(* IEC 61131-3 sources: moqui-plc/iec61131/moqui/framework/src/main/org/moqui/device, 53 files *)

(* ---- ActuatorActuationType.dut ---- *)
(*#-#-#-#-#-#-#-#-#-#---Declaration---#-#-#-#-#-#-#-#-#-#-#-#-#*)

{attribute 'qualified_only'}
{attribute 'strict'}
TYPE ActuatorActuationType : (
    SingleActuation := 0, (* Single Actuation: Uses enable output only *)
    DoubleActuation, (* Double Actuation: enable/disable are pulses *)
    DoubleActuationNoRetain (* Double Actuation: enable/disable are levels *)
); END_TYPE

(* ---- ActuatorActuationType.st ---- *)
TYPE ActuatorActuationType : (
    SingleActuation := 0, (* Single Actuation: Uses enable output only *)
    DoubleActuation, (* Double Actuation: enable/disable are pulses *)
    DoubleActuationNoRetain (* Double Actuation: enable/disable are levels *)
); END_TYPE

(* ---- ActuatorFeedbackType.dut ---- *)
(*#-#-#-#-#-#-#-#-#-#---Declaration---#-#-#-#-#-#-#-#-#-#-#-#-#*)

{attribute 'qualified_only'}
{attribute 'strict'}
TYPE ActuatorFeedbackType : (
	WithoutFeedback := 0, (* No feedback *)
    SingleDisableFeedback, (* Single Deactivation Feedback: Only disabledSensor *)
    SingleEnableFeedback, (* Single Activation Feedback: Only enabledSensor *)
	DoubleFeedback (* Double Feedback: Both sensors *)
); END_TYPE

(* ---- ActuatorFeedbackType.st ---- *)
TYPE ActuatorFeedbackType : (
	WithoutFeedback := 0, (* No feedback *)
    SingleDisableFeedback, (* Single Deactivation Feedback: Only disabledSensor *)
    SingleEnableFeedback, (* Single Activation Feedback: Only enabledSensor *)
	DoubleFeedback (* Double Feedback: Both sensors *)
); END_TYPE

(* ---- ActuatorGroupAutochange.dut ---- *)
(*#-#-#-#-#-#-#-#-#-#---Declaration---#-#-#-#-#-#-#-#-#-#-#-#-#*)

{attribute 'qualified_only'}
{attribute 'strict'}
(*
 * Selects the mode used to trigger a priority-order rotation (autochange).
 * Corresponds to ABB ACH580 parameter 76.70 Autochange.
 *)
TYPE ActuatorGroupAutochange : (
    None := 0, (* Autochange disabled; priority order is fixed *)
    EvenWear, (* Rotate when run-hour imbalance > maxWearImbalance (76.72) *)
    FixedInterval, (* Rotate every autochangeInterval when demand ≤ autochangeLevel (76.71) *)
    ExternalTrigger, (* Rotate on rising edge of autochangeTrigger when demand ≤ autochangeLevel *)
    AllStopped (* Rotate whenever the group stops (all actuators off) *)
); END_TYPE

(* ---- ActuatorGroupAutochange.st ---- *)
(*
 * Selects the mode used to trigger a priority-order rotation (autochange).
 * Corresponds to ABB ACH580 parameter 76.70 Autochange.
 *)
TYPE ActuatorGroupAutochange : (
    None := 0, (* Autochange disabled; priority order is fixed *)
    EvenWear, (* Rotate when run-hour imbalance > maxWearImbalance (76.72) *)
    FixedInterval, (* Rotate every autochangeInterval when demand <= autochangeLevel (76.71) *)
    ExternalTrigger, (* Rotate on rising edge of autochangeTrigger when demand <= autochangeLevel *)
    AllStopped (* Rotate whenever the group stops (all actuators off) *)
); END_TYPE

(* ---- ActuatorGroupStatus.dut ---- *)
(*#-#-#-#-#-#-#-#-#-#---Declaration---#-#-#-#-#-#-#-#-#-#-#-#-#*)

{attribute 'qualified_only'}
{attribute 'strict'}
TYPE ActuatorGroupStatus : (
    Disabled := 0, (* No actuators running; group not active *)
    Running, (* Active: demand-driven start/stop in progress *)
    Stopping, (* Transitional: shutting down all running actuators *)
    Autochange (* Transitional: rotating the priority order (stop old / start new) *)
); END_TYPE

(* ---- ActuatorGroupStatus.st ---- *)
TYPE ActuatorGroupStatus : (
    Disabled := 0, (* No actuators running; group not active *)
    Running, (* Active: demand-driven start/stop in progress *)
    Stopping, (* Transitional: shutting down all running actuators *)
    Autochange (* Transitional: rotating the priority order (stop old / start new) *)
); END_TYPE

(* ---- ActuatorModel.dut ---- *)
(*#-#-#-#-#-#-#-#-#-#---Declaration---#-#-#-#-#-#-#-#-#-#-#-#-#*)

{attribute 'qualified_only'}
TYPE ActuatorModel : (
	ABBACH580, (* ABB ACH580 *)
	CTM700, (* Control Techniques CM700 *)
	DanfossFC102, (* Danfoss FC102 *)
	ABBPSTX (* ABB PSTX SoftStarter *)
	(* etc. *)
); END_TYPE

(* ---- ActuatorStatus.dut ---- *)
(*#-#-#-#-#-#-#-#-#-#---Declaration---#-#-#-#-#-#-#-#-#-#-#-#-#*)

{attribute 'qualified_only'}
{attribute 'strict'}
TYPE ActuatorStatus : (
	Disabled := 0, (* Stable *)
	EnablePhase, (* Unstable *)
	Enabled, (* Stable *)
	DisablePhase (* Unstable *)
); END_TYPE

(* ---- ActuatorStatus.st ---- *)
TYPE ActuatorStatus : (
	Disabled := 0, (* Stable *)
	EnablePhase, (* Unstable *)
	Enabled, (* Stable *)
	DisablePhase (* Unstable *)
); END_TYPE

(* ---- ActuatorType.dut ---- *)
(*#-#-#-#-#-#-#-#-#-#---Declaration---#-#-#-#-#-#-#-#-#-#-#-#-#*)

{attribute 'qualified_only'}
{attribute 'strict'}
TYPE ActuatorType : (
  OnOff := 0, (* Fallback value *)
  Contactor,
  SoftStarter,
  Vfd, (* Frequency converter / Inverter drive *)
  PneumaticCylinder,
  PneumaticValve,
  HydraulicCylinder,
  HydraulicValve,
  Damper,
  SolenoidValve
  (* etc. *)
); END_TYPE

(* ---- ActuatorType.st ---- *)
TYPE ActuatorType : (
  OnOff := 0, (* Fallback value *)
  Contactor,
  SoftStarter,
  Vfd, (* Frequency converter / Inverter drive *)
  PneumaticCylinder,
  PneumaticValve,
  HydraulicCylinder,
  HydraulicValve,
  Damper,
  SolenoidValve
  (* etc. *)
); END_TYPE

(* ---- DeviceConfigCmdType.dut ---- *)
(*#-#-#-#-#-#-#-#-#-#---Declaration---#-#-#-#-#-#-#-#-#-#-#-#-#*)

{attribute 'qualified_only'}
{attribute 'strict'}
(* After each creation, saving or deletion of device config it will be necessary to reload the config list with the Init command. *)
TYPE DeviceConfigCmdType : (
    Init := 0, (* Init the recipe management component *)
	Create,
    Save,
	Load,
	Delete,
	Reset
); END_TYPE

(* ---- DeviceConfigCmdType.st ---- *)
(* After each creation, saving or deletion of device config it will be necessary to reload the config list with the Init command. *)
TYPE DeviceConfigCmdType : (
    Init := 0, (* Init the recipe management component *)
	Create,
    Save,
	Load,
	Delete,
	Reset
); END_TYPE

(* ---- DeviceConfigMgmtStatus.dut ---- *)
(*#-#-#-#-#-#-#-#-#-#---Declaration---#-#-#-#-#-#-#-#-#-#-#-#-#*)

{attribute 'qualified_only'}
{attribute 'strict'}
TYPE DeviceConfigMgmtStatus : (
    Idle,
	Init,
	Resetting,
    Check,
    Load,
    WaitLoad,
    WaitProcessing,
    IncrementIndex,
    Completed,
    Error
); END_TYPE

(* ---- DriveControlWord.dut ---- *)
(*#-#-#-#-#-#-#-#-#-#---Declaration---#-#-#-#-#-#-#-#-#-#-#-#-#*)

{attribute 'qualified_only'}
(* Drive control words *)
(* Relevant control word for start, stop and reset commands *)
TYPE DriveControlWord : (
	(* ABB ACS580, ACH580 drive *)
	ABBACH580Reset := 1278,
	ABBACH580Stop := 1150,
	ABBACH580Start := 1151,
	(* Control Techniques M600 drive *)
	CTM600Reset := 111,
	CTM600Stop := 112,
	CTM600Start := 113,
	(* Danfoss FC102 drive *)
	DanfossFC102Reset := 121,
	DanfossFC102Stop := 122,
	DanfossFC102Start := 123
); END_TYPE

(* ---- DriveControlWord.st ---- *)
(* Drive control words *)
(* Relevant control word for start, stop and reset commands *)
TYPE DriveControlWord : (
	(* ABB ACS580, ACH580 drive *)
	ABBACH580Reset := 1278,
	ABBACH580Stop := 1150,
	ABBACH580Start := 1151,
	(* Control Techniques M600 drive *)
	CTM600Reset := 111,
	CTM600Stop := 112,
	CTM600Start := 113,
	(* Danfoss FC102 drive *)
	DanfossFC102Reset := 121,
	DanfossFC102Stop := 122,
	DanfossFC102Start := 123
); END_TYPE

(* ---- EdgeTriggerStatus.dut ---- *)
(*#-#-#-#-#-#-#-#-#-#---Declaration---#-#-#-#-#-#-#-#-#-#-#-#-#*)

{attribute 'qualified_only'}
{attribute 'strict'}
TYPE EdgeTriggerStatus : (
	Dormant := 0,
	Executing,
	Done,
	Aborting,
	Aborted,
	Resetting,
	Error
); END_TYPE

(* ---- EdgeTriggerStatus.st ---- *)
TYPE EdgeTriggerStatus : (
	Dormant := 0,
	Executing,
	Done,
	Aborting,
	Aborted,
	Resetting,
	Error
); END_TYPE

(* ---- FieldbusProtocol.dut ---- *)
(*#-#-#-#-#-#-#-#-#-#---Declaration---#-#-#-#-#-#-#-#-#-#-#-#-#*)

{attribute 'qualified_only'}
TYPE FieldbusProtocol : (
	ModbusTCP,
	ModbusRTU,
	EthernetIP,
	Profinet,
	CanOpen
); END_TYPE

(* ---- FieldbusProtocol.st ---- *)
TYPE FieldbusProtocol : (
	ModbusTCP,
	ModbusRTU,
	EthernetIP,
	Profinet,
	CanOpen
); END_TYPE

(* ---- LevelCtrlStatus.dut ---- *)
(*#-#-#-#-#-#-#-#-#-#---Declaration---#-#-#-#-#-#-#-#-#-#-#-#-#*)

{attribute 'qualified_only'}
{attribute 'strict'}
TYPE LevelCtrlStatus : (
	Dormant := 0,
	Executing,
	Done,
	Aborting,
	Resetting,
	Error
); END_TYPE

(* ---- LevelCtrlStatus.st ---- *)
TYPE LevelCtrlStatus : (
	Dormant := 0,
	Executing,
	Done,
	Aborting,
	Resetting,
	Error
); END_TYPE

(* ---- OperatingMode.dut ---- *)
(*#-#-#-#-#-#-#-#-#-#---Declaration---#-#-#-#-#-#-#-#-#-#-#-#-#*)

{attribute 'qualified_only'}
{attribute 'strict'}
TYPE OperatingMode : (
	Init := 1,
	Run
); END_TYPE

(* ---- OperatingMode.st ---- *)
TYPE OperatingMode : (
	Init := 1,
	Run
); END_TYPE

(* ---- RampType.dut ---- *)
(*#-#-#-#-#-#-#-#-#-#---Declaration---#-#-#-#-#-#-#-#-#-#-#-#-#*)

{attribute 'qualified_only'}
TYPE RampType : (
    Linear, // Linear ramp.
    SShaped, // S-Shaped ramp.
    Exponential, // Exponential ramp
    Custom // Custom-defined ramp function
); END_TYPE

(* ---- SpeedSetpointLevel.dut ---- *)
(*#-#-#-#-#-#-#-#-#-#---Declaration---#-#-#-#-#-#-#-#-#-#-#-#-#*)

{attribute 'qualified_only'}
{attribute 'strict'}
(* Constants are defined to represent the different speed levels required by a motor.
 * Alternatively, the speed setpoint/reference can be defined as a continuous analog output.
 * It is possible to apply the same logic to other variables such as:
 *     acceleration/deceleration, torque, etc.
 *)
TYPE SpeedSetpointLevel : (
	ZeroSpeed := 0,
	NominalSpeed,
	MinSpeed,
	MaxSpeed,
	JoggingSpeed,
	SafelyLimitedSpeed
	(* etc. *)
); END_TYPE

(* ---- SpeedSetpointLevel.st ---- *)
(* Constants are defined to represent the different speed levels required by a motor.
 * Alternatively, the speed setpoint/reference can be defined as a continuous analog output.
 * It is possible to apply the same logic to other variables such as:
 *     acceleration/deceleration, torque, etc.
 *)
TYPE SpeedSetpointLevel : (
	ZeroSpeed := 0,
	NominalSpeed,
	MinSpeed,
	MaxSpeed,
	JoggingSpeed,
	SafelyLimitedSpeed
	(* etc. *)
); END_TYPE

(* ---- processAnalogInput.pou ---- *)
(*#-#-#-#-#-#-#-#-#-#---Declaration---#-#-#-#-#-#-#-#-#-#-#-#-#*)

(* Conversion and processing of a physical input signal into a logical parameter *)
FUNCTION processAnalogInput : REAL
VAR_INPUT
	physicalValue : WORD;
	minPhysicalValue, maxPhysicalValue : WORD;
	minValue, maxValue : REAL;
	offset : REAL := 0;
	scalingFactor : REAL := 1;
	significantDigits : INT := 2;
END_VAR
VAR
	inputValue : REAL;
END_VAR

(*#-#-#-#-#-#-#-#-#-#---Implementation---#-#-#-#-#-#-#-#-#-#-#-#-#*)

inputValue := TO_REAL(physicalValue);
inputValue := scale(inputValue, minPhysicalValue, maxPhysicalValue, minValue, maxValue);
inputValue := inputValue * scalingFactor + offset;
inputValue := LIMIT(minValue, inputValue, maxValue);

IF significantDigits = 0 THEN
	inputValue := truncReal(inputValue, significantDigits);
ELSIF significantDigits > 0 THEN
	inputValue := round(inputValue, significantDigits);
END_IF;

processAnalogInput := TO_REAL(inputValue);

(* ---- processAnalogInput.st ---- *)
(* Conversion and processing of a physical input signal into a logical parameter *)
FUNCTION processAnalogInput : REAL
	VAR_INPUT
		physicalValue : WORD;
		minPhysicalValue, maxPhysicalValue : WORD;
		minValue, maxValue : REAL;
		offset : REAL := 0;
		scalingFactor : REAL := 1;
		significantDigits : INT := 2;
	END_VAR
	VAR
		inputValue : REAL;
	END_VAR

	inputValue := TO_REAL(physicalValue);
	inputValue := scale(inputValue, minPhysicalValue, maxPhysicalValue, minValue, maxValue);
	inputValue := inputValue * scalingFactor + offset;
	inputValue := LIMIT(minValue, inputValue, maxValue);

	IF significantDigits = 0 THEN
		inputValue := truncReal(inputValue, significantDigits);
	ELSIF significantDigits > 0 THEN
		inputValue := round(inputValue, significantDigits);
	END_IF;

	processAnalogInput := TO_REAL(inputValue);
	END_FUNCTION

(* ---- processAnalogOutput.pou ---- *)
(*#-#-#-#-#-#-#-#-#-#---Declaration---#-#-#-#-#-#-#-#-#-#-#-#-#*)

(* Conversion and processing of a logical parameter into a physical signal *)
FUNCTION processAnalogOutput : BOOL
VAR_INPUT
	parameterValue : REAL;
	minPhysicalValue, maxPhysicalValue : WORD;
	minValue, maxValue : REAL;
	offset : REAL := 0;
	scalingFactor : REAL := 1;
	significantDigits : INT := 2;
	littleEndian : BOOL := TRUE;
END_VAR
VAR_OUTPUT
	byteAnalogOutput : BYTE;
	wordAnalogOutput : WORD;
	dWordAnalogOutput : DWORD;
END_VAR
VAR
	outputValue : REAL;
END_VAR

(*#-#-#-#-#-#-#-#-#-#---Implementation---#-#-#-#-#-#-#-#-#-#-#-#-#*)

processAnalogOutput := FALSE;

outputValue := (parameterValue - offset) / scalingFactor;
outputValue := LIMIT(minValue, outputValue, maxValue);
outputValue := scale(outputValue, minValue, maxValue, minPhysicalValue, maxPhysicalValue);

IF significantDigits = 0 THEN
	outputValue := truncReal(outputValue, significantDigits);
ELSIF significantDigits > 0 THEN
	outputValue := round(outputValue, significantDigits);
END_IF;

byteAnalogOutput := TO_BYTE(outputValue);

IF littleEndian THEN
	wordAnalogOutput := TO_WORD(outputValue);
	dWordAnalogOutput := TO_DWORD(outputValue);
ELSE
	wordAnalogOutput := swapWordEndian(TO_WORD(outputValue));
	dWordAnalogOutput := swapDWordEndian(TO_DWORD(outputValue));
END_IF;

processAnalogOutput := TRUE;

(* ---- processAnalogOutput.st ---- *)
(* Conversion and processing of a logical parameter into a physical signal *)
FUNCTION processAnalogOutput : BOOL
	VAR_INPUT
		parameterValue : REAL;
		minPhysicalValue, maxPhysicalValue : WORD;
		minValue, maxValue : REAL;
		offset : REAL := 0;
		scalingFactor : REAL := 1;
		significantDigits : INT := 2;
		littleEndian : BOOL := TRUE;
	END_VAR
	VAR_OUTPUT
		byteAnalogOutput : BYTE;
		wordAnalogOutput : WORD;
		dWordAnalogOutput : DWORD;
	END_VAR
	VAR
		outputValue : REAL;
	END_VAR

	processAnalogOutput := FALSE;

	outputValue := (parameterValue - offset) / scalingFactor;
	outputValue := LIMIT(minValue, outputValue, maxValue);
	outputValue := scale(outputValue, minValue, maxValue, minPhysicalValue, maxPhysicalValue);

	IF significantDigits = 0 THEN
		outputValue := truncReal(outputValue, significantDigits);
	ELSIF significantDigits > 0 THEN
		outputValue := round(outputValue, significantDigits);
	END_IF;

	byteAnalogOutput := TO_BYTE(outputValue);

	IF littleEndian THEN
		wordAnalogOutput := TO_WORD(outputValue);
		dWordAnalogOutput := TO_DWORD(outputValue);
	ELSE
		wordAnalogOutput := swapWordEndian(TO_WORD(outputValue));
		dWordAnalogOutput := swapDWordEndian(TO_DWORD(outputValue));
	END_IF;

	processAnalogOutput := TRUE;
	END_FUNCTION

(* ---- processCyclicInFieldbusData.pou ---- *)
(*#-#-#-#-#-#-#-#-#-#---Declaration---#-#-#-#-#-#-#-#-#-#-#-#-#*)

(* Mapping of bits of the fieldbus status word to the basic actuator inputs *)
FUNCTION processCyclicInFieldbusData : BOOL
VAR_INPUT
	model : ActuatorModel;
	fieldbus : FieldbusProtocol;
	statusWord : WORD;
END_VAR
VAR_OUTPUT
	enabledSensor : BOOL := FALSE;
	disabledSensor : BOOL := FALSE;
	externalFault : BOOL := FALSE;
END_VAR

(*#-#-#-#-#-#-#-#-#-#---Implementation---#-#-#-#-#-#-#-#-#-#-#-#-#*)

processCyclicInFieldbusData := FALSE;

CASE model OF
	ActuatorModel.ABBACH580 :
		(* Set parameters based on the drive statusWord interpretation *)
		enabledSensor := statusWord.0 AND statusWord.1 AND statusWord.2;
		disabledSensor := NOT statusWord.0 OR NOT statusWord.1 OR NOT statusWord.2;
		externalFault := statusWord.3 OR statusWord.4 OR statusWord.5 OR statusWord.6 OR statusWord.9;
	ActuatorModel.CTM700 :
		(* etc. *)
	ActuatorModel.DanfossFc102 :
		(* etc. *)
	ELSE
		RETURN;
END_CASE;

processCyclicInFieldbusData := TRUE;

(* ---- processCyclicInFieldbusData.st ---- *)
(* Mapping of bits of the fieldbus status word to the basic actuator inputs *)
FUNCTION processCyclicInFieldbusData : BOOL
	VAR_INPUT
		model : ActuatorModel;
		fieldbus : FieldbusProtocol;
		statusWord : WORD;
	END_VAR
	VAR_OUTPUT
		enabledSensor : BOOL := FALSE;
		disabledSensor : BOOL := FALSE;
		externalFault : BOOL := FALSE;
	END_VAR

	processCyclicInFieldbusData := FALSE;

	CASE model OF
		ActuatorModel.ABBACH580 :
			(* Set parameters based on the drive statusWord interpretation *)
			enabledSensor := statusWord.0 AND statusWord.1 AND statusWord.2;
			disabledSensor := NOT statusWord.0 OR NOT statusWord.1 OR NOT statusWord.2;
			externalFault := statusWord.3 OR statusWord.4 OR statusWord.5 OR statusWord.6 OR statusWord.9;
		ActuatorModel.CTM700 :
			(* etc. *)
		ActuatorModel.DanfossFc102 :
			(* etc. *)
		ELSE
			RETURN;
	END_CASE;

	processCyclicInFieldbusData := TRUE;
	END_FUNCTION

(* ---- processCyclicOutFieldbusData.pou ---- *)
(*#-#-#-#-#-#-#-#-#-#---Declaration---#-#-#-#-#-#-#-#-#-#-#-#-#*)

(* Mapping of basic actuator outputs to bits of the fieldbus control word *)
FUNCTION processCyclicOutFieldbusData : BOOL
VAR_INPUT
	model : ActuatorModel;
	fieldbus : FieldbusProtocol;
	enable : BOOL;
	disable : BOOL;
	reset : BOOL;
	(*
	 * Declare this enum only if you use finite set of levels for the speed setpoint or reference.
	 * They could be mapped to the drive's control word user bits.
	 * The same approach can be used for other drive parameters such as frequency,
     * acceleration/deceleration, torque, estimated position, etc... based on available user bits.
	 *)
	(* speedSetpoint : SpeedSetpointLevel := SpeedSetpointLevel.ZeroSpeed; *)
END_VAR
VAR_OUTPUT
	controlWord : WORD;
END_VAR

(*#-#-#-#-#-#-#-#-#-#---Implementation---#-#-#-#-#-#-#-#-#-#-#-#-#*)

processCyclicOutFieldbusData := FALSE;

IF enable THEN
	CASE model OF
		ActuatorModel.ABBACH580 :
			controlWord := TO_WORD(DriveControlWord.ABBACH580Start);
		ActuatorModel.CTM700 :
			controlWord := TO_WORD(DriveControlWord.CTM600Start);
		ActuatorModel.DanfossFc102 :
			controlWord := TO_WORD(DriveControlWord.DanfossFC102Start);
		ELSE
			RETURN;
	END_CASE;
ELSE
	CASE model OF
		ActuatorModel.ABBACH580 :
			controlWord := TO_WORD(DriveControlWord.ABBACH580Stop);
		ActuatorModel.CTM700 :
			controlWord := TO_WORD(DriveControlWord.CTM600Stop);
		ActuatorModel.DanfossFc102 :
			controlWord := TO_WORD(DriveControlWord.DanfossFC102Stop);
		ELSE
			RETURN;
	END_CASE;
END_IF;

IF reset THEN
	CASE model OF
		ActuatorModel.ABBACH580 :
			controlWord := TO_WORD(DriveControlWord.ABBACH580Reset);
		ActuatorModel.CTM700 :
			controlWord := TO_WORD(DriveControlWord.CTM600Reset);
		ActuatorModel.DanfossFc102 :
			controlWord := TO_WORD(DriveControlWord.DanfossFC102Reset);
		ELSE
			RETURN;
	END_CASE;
END_IF;

(*
(*
 * Example of speed selection for drive with finite set of levels for speed.
 * Use index access to change the drive's control word user bits (see below).
 * It is possible to apply the same logic to other variables such as:
 *     frequency, acceleration/deceleration, torque, estimated position, etc.
 *)
CASE speedSetpoint OF
	SpeedSetpointLevel.ZeroSpeed :
		controlWord.12 := 0;
		controlWord.13 := 0;
		controlWord.14 := 0;
	SpeedSetpointLevel.MinSpeed :
		controlWord.12 := 1;
		controlWord.13 := 0;
		controlWord.14 := 0;
	SpeedSetpointLevel.NominalSpeed :
		controlWord.12 := 0;
		controlWord.13 := 1;
		controlWord.14 := 0;
	SpeedSetpointLevel.MaxSpeed :
		controlWord.12 := 1;
		controlWord.13 := 1;
		controlWord.14 := 0;
	SpeedSetpointLevel.JoggingSpeed :
		controlWord.12 := 0;
		controlWord.13 := 0;
		controlWord.14 := 1;
	SpeedSetpointLevel.SafelyLimitedSpeed :
		controlWord.12 := 1;
		controlWord.13 := 0;
		controlWord.14 := 1;
END_CASE;
*)

processCyclicOutFieldbusData := TRUE;

(* ---- processCyclicOutFieldbusData.st ---- *)
(* Mapping of basic actuator outputs to bits of the fieldbus control word *)
FUNCTION processCyclicOutFieldbusData : BOOL
	VAR_INPUT
		model : ActuatorModel;
		fieldbus : FieldbusProtocol;
		enable : BOOL;
		disable : BOOL;
		reset : BOOL;
		(*
		 * Declare this enum only if you use finite set of levels for the speed setpoint or reference.
		 * They could be mapped to the drive's control word user bits.
		 * The same approach can be used for other drive parameters such as frequency,
	     * acceleration/deceleration, torque, estimated position, etc... based on available user bits.
		 *)
		(* speedSetpoint : SpeedSetpointLevel := SpeedSetpointLevel.ZeroSpeed; *)
	END_VAR
	VAR_OUTPUT
		controlWord : WORD;
	END_VAR

	processCyclicOutFieldbusData := FALSE;

	IF enable THEN
		CASE model OF
			ActuatorModel.ABBACH580 :
				controlWord := TO_WORD(DriveControlWord.ABBACH580Start);
			ActuatorModel.CTM700 :
				controlWord := TO_WORD(DriveControlWord.CTM600Start);
			ActuatorModel.DanfossFc102 :
				controlWord := TO_WORD(DriveControlWord.DanfossFC102Start);
			ELSE
				RETURN;
		END_CASE;
	ELSE
		CASE model OF
			ActuatorModel.ABBACH580 :
				controlWord := TO_WORD(DriveControlWord.ABBACH580Stop);
			ActuatorModel.CTM700 :
				controlWord := TO_WORD(DriveControlWord.CTM600Stop);
			ActuatorModel.DanfossFc102 :
				controlWord := TO_WORD(DriveControlWord.DanfossFC102Stop);
			ELSE
				RETURN;
		END_CASE;
	END_IF;

	IF reset THEN
		CASE model OF
			ActuatorModel.ABBACH580 :
				controlWord := TO_WORD(DriveControlWord.ABBACH580Reset);
			ActuatorModel.CTM700 :
				controlWord := TO_WORD(DriveControlWord.CTM600Reset);
			ActuatorModel.DanfossFc102 :
				controlWord := TO_WORD(DriveControlWord.DanfossFC102Reset);
			ELSE
				RETURN;
		END_CASE;
	END_IF;

	(*
	(*
	 * Example of speed selection for drive with finite set of levels for speed.
	 * Use index access to change the drive's control word user bits (see below).
	 * It is possible to apply the same logic to other variables such as:
	 *     frequency, acceleration/deceleration, torque, estimated position, etc.
	 *)
	CASE speedSetpoint OF
		SpeedSetpointLevel.ZeroSpeed :
			controlWord.12 := 0;
			controlWord.13 := 0;
			controlWord.14 := 0;
		SpeedSetpointLevel.MinSpeed :
			controlWord.12 := 1;
			controlWord.13 := 0;
			controlWord.14 := 0;
		SpeedSetpointLevel.NominalSpeed :
			controlWord.12 := 0;
			controlWord.13 := 1;
			controlWord.14 := 0;
		SpeedSetpointLevel.MaxSpeed :
			controlWord.12 := 1;
			controlWord.13 := 1;
			controlWord.14 := 0;
		SpeedSetpointLevel.JoggingSpeed :
			controlWord.12 := 0;
			controlWord.13 := 0;
			controlWord.14 := 1;
		SpeedSetpointLevel.SafelyLimitedSpeed :
			controlWord.12 := 1;
			controlWord.13 := 0;
			controlWord.14 := 1;
	END_CASE;
	*)

	processCyclicOutFieldbusData := TRUE;
	END_FUNCTION

(* ---- processMotorStarterInData.pou ---- *)
(*#-#-#-#-#-#-#-#-#-#---Declaration---#-#-#-#-#-#-#-#-#-#-#-#-#*)

(* Mapping inputs of a manual motor starter, motor protection circuit breakers (MPCBs)
 * and contactors, to the basic actuator inputs. *)
FUNCTION processMotorStarterInData : BOOL
VAR_INPUT
	contactorAuxiliaryContact : BOOL;
	motorStarterSignallingContact : BOOL;
	motorStarterShuntTrip : BOOL;
END_VAR
VAR_OUTPUT
	enabledSensor : BOOL := FALSE;
	disabledSensor : BOOL := FALSE;
	externalFault : BOOL := FALSE;
END_VAR

(*#-#-#-#-#-#-#-#-#-#---Implementation---#-#-#-#-#-#-#-#-#-#-#-#-#*)

processMotorStarterInData := FALSE;

(* Set parameters based on the motor starter signals interpretation *)
enabledSensor := contactorAuxiliaryContact;
disabledSensor := NOT contactorAuxiliaryContact;
externalFault := NOT contactorAuxiliaryContact OR motorStarterShuntTrip;

processMotorStarterInData := TRUE;

(* ---- processMotorStarterInData.st ---- *)
(* Mapping inputs of a manual motor starter, motor protection circuit breakers (MPCBs)
 * and contactors, to the basic actuator inputs. *)
FUNCTION processMotorStarterInData : BOOL
	VAR_INPUT
		contactorAuxiliaryContact : BOOL;
		motorStarterSignallingContact : BOOL;
		motorStarterShuntTrip : BOOL;
	END_VAR
	VAR_OUTPUT
		enabledSensor : BOOL := FALSE;
		disabledSensor : BOOL := FALSE;
		externalFault : BOOL := FALSE;
	END_VAR

	processMotorStarterInData := FALSE;

	(* Set parameters based on the motor starter signals interpretation *)
	enabledSensor := contactorAuxiliaryContact;
	disabledSensor := NOT contactorAuxiliaryContact;
	externalFault := NOT contactorAuxiliaryContact OR motorStarterShuntTrip;

	processMotorStarterInData := TRUE;
	END_FUNCTION

(* ---- Actuator.pou ---- *)
(*#-#-#-#-#-#-#-#-#-#---Declaration---#-#-#-#-#-#-#-#-#-#-#-#-#*)

{attribute 'no_assign'}
(*
 * Generic binary actuator control system/automata, including mechanisms diagnostics.
 * In nominal conditions, a binary actuator has only two stable equilibrium states: Disabled, Enabled.
 * It also has two unstable transient states: EnablePhase, DisablePhase.
 * The remainder are inadmissible states that must be detected based on timing conditions.
 * Nominal trajectory in the state space, i.e. the evolution of the state in nominal working conditions:
 *     Disabled --> EnablePhase --> Enabled --> DisabledPhase --> back to Disabled
 * Admissible states transitions:
 *     EnablePhase --> DisablePhase, DisablePhase --> EnablePhase
 *
 * Handshake-based actuator control via VAR_IN_OUT.
 * This function block utilizes a Request/Acknowledge (Handshake) mechanism
 * through VAR_IN_OUT variables to manage asynchronous device operations.
 *
 * Usage Logic:
 *  - The caller sets the 'enableRequest' variable to TRUE to initiate the process.
 *  - The FB monitors this variable and attempts to enable the physical device.
 *  - Upon successful activation, the FB internally resets 'enableRequest' to FALSE.
 *
 * Sequencing and diagnostics:
 *  - Sequencing: By monitoring the falling edge of the request variable (Request -> FALSE),
 *    the application logic can deterministically trigger the next step in a sequence
 *    without relying on timers or intermediate state flags.
 *  - Real-Time diagnostics: If the request remains TRUE beyond a defined timeout period,
 *    it indicates a failure in the handshake (e.g., hardware interlock or communication error).
 *    This allows for immediate error detection (machineError) and prevents the
 *    sequence from advancing in an unsafe state.
 *
 * Note:
 * Since the variable is passed by reference (VAR_IN_OUT), both the caller and
 * the FB share the same memory location, ensuring atomic-like synchronization of the command status.
 * This mechanism is used to allow sequencing of the start/stop phases in the presence of a group of devices.
 *
 *)
FUNCTION_BLOCK Actuator
(* Request/Ack commands *)
VAR_IN_OUT
    enableRequest : BOOL;
    disableRequest : BOOL;
END_VAR
VAR_INPUT
	(* Actuator metadata for logging purpose *)
	actuatorId : STRING;
	actuatorName : STRING;
  	actuationType : ActuatorActuationType;
	feedbackType : ActuatorFeedbackType;
	model : ActuatorModel;
    operationType : OperatingMode := OperatingMode.Run;
	(* Clock for diagnosis and fault detection under static and dynamic conditions *)
    clock : BOOL;
	(* Time limit for the enable/disable phase *)
    enableTime : UINT;
    disableTime : UINT;
	(* Preset/Reset *)
    enablePreset : BOOL := FALSE;
    (* Enable diagnostics *)
    diagnosticsEnable : BOOL := TRUE;
END_VAR
VAR_INPUT
	(* Actuator status sensors *)
    enabledSensor : BOOL;
    disabledSensor : BOOL;
	(* External fault signal (e.g. motor branch-circuit protection, thermal relay) *)
	externalFault : BOOL;
	(* Optional parameters  *)
  	ref : REAL;
  	feedback : REAL;
END_VAR
VAR_OUTPUT
	(* Diagnostics and fault signals *)
    fault : BOOL;
    actuatorFault : BOOL;
    enabledSensorFault : BOOL;
    disabledSensorFault : BOOL;
    notInitialized : BOOL;
	(* Logger name for centralized signal management *)
	loggerName : STRING;
END_VAR
VAR_OUTPUT
	(* Output signals *)
	enable : BOOL;
    disable : BOOL;
END_VAR
VAR
    status : ActuatorStatus;
    timer : UINT;
    timeout : BOOL;
	(* Internal logical feedback signals (derived from external sensors and/or state + timeout). *)
	enabled : BOOL;
	disabled : BOOL;
	(* Logger facade *)
	logger : LoggerFacade;
END_VAR

(*#-#-#-#-#-#-#-#-#-#---Implementation---#-#-#-#-#-#-#-#-#-#-#-#-#*)

(* Initialization handler *)
IF operationType = OperatingMode.Init THEN
	(* Args validation *)
	IF (actuatorId = '' AND actuatorName = '') THEN
		notInitialized := TRUE;
		RETURN;
	END_IF;

	(* Logger facade init *)
	loggerName := concat(concat(concat(actuatorName, '['), actuatorId), ']');
	logger.enable := TRUE; logger.loggerName := loggerName;

	logger(message := 'Actuator initialization.', level := LogLevel.DEBUG);

	(* Pre-elaborations for initialization (polymorphism on feedback typology). *)
	CASE feedbackType OF
		ActuatorFeedbackType.DoubleFeedback :
			enabled := enabledSensor;
			disabled := disabledSensor;

		ActuatorFeedbackType.SingleEnableFeedback :
			enabled := enabledSensor;
			disabled := NOT enabled;

		ActuatorFeedbackType.SingleDisableFeedback :
			disabled := disabledSensor;
			enabled := NOT disabled;

		ActuatorFeedbackType.WithoutFeedback :
			enabled := enablePreset;
			disabled := NOT enabled;
	END_CASE;

	enableRequest := FALSE;
	disableRequest := FALSE;

    IF enablePreset THEN
		logger(message := 'Actuator preset to enabled status.', level := LogLevel.DEBUG);
		enable := TRUE;
		timer := enableTime;

		IF enabled THEN
			status := ActuatorStatus.Enabled;
			notInitialized := FALSE;
		ELSE
			status := ActuatorStatus.EnablePhase;
            notInitialized := TRUE;
		END_IF;
    ELSE
		logger(message := 'Actuator preset to disabled status.', level := LogLevel.DEBUG);
		enable := FALSE;
		timer := disableTime;

		IF disabled THEN
            status := ActuatorStatus.Disabled;
            notInitialized := FALSE;
        ELSE
            status := ActuatorStatus.DisablePhase;
            notInitialized := TRUE;
        END_IF;
	END_IF;
END_IF;

IF notInitialized THEN logger(message := 'Actuator not initialized.', level := LogLevel.ERROR); END_IF;

logger(message := 'Running actuator.', level := LogLevel.DEBUG);

(* Clock handler for diagnosis oriented timing *)
IF clock AND (timer > 0) THEN
    timer := timer - 1;
END_IF;

(* Timeout computation *)
timeout := (timer = 0);

(* Pre-elaborations for feedback polymorphism. *)
CASE feedbackType OF
	ActuatorFeedbackType.DoubleFeedback :
		enabled := enabledSensor;
		disabled := disabledSensor;

	ActuatorFeedbackType.SingleDisableFeedback :
		disabled := disabledSensor;
		enabled := (NOT disabled) AND ((status = ActuatorStatus.Enabled)
			OR ((status = ActuatorStatus.EnablePhase) AND timeout));

	ActuatorFeedbackType.SingleEnableFeedback :
		enabled := enabledSensor;
		disabled := (NOT enabled) AND ((status = ActuatorStatus.Disabled)
			OR ((status = ActuatorStatus.DisablePhase) AND timeout));

	ActuatorFeedbackType.WithoutFeedback :
		enabled := (status = ActuatorStatus.Enabled) OR ((status = ActuatorStatus.EnablePhase) AND timeout);
		disabled := (status = ActuatorStatus.Disabled) OR ((status = ActuatorStatus.DisablePhase) AND timeout);
END_CASE;

(* Generic actuator FSM implementation. *)
CASE status OF
	ActuatorStatus.Disabled :
		logger(message := 'Actuator disabled.', level := LogLevel.DEBUG);
		disableRequest := FALSE;

		IF enableRequest THEN
			logger(message := 'The actuator received an enable request.', level := LogLevel.DEBUG);
			enable := TRUE;
			timer := enableTime;
			status := ActuatorStatus.EnablePhase;
		END_IF;

	ActuatorStatus.EnablePhase :
		logger(message := 'Actuator in the enabling phase.', level := LogLevel.DEBUG);

		(* Admissible transition: EnablePhase --> DisablePhase *)
		IF disableRequest THEN
			logger(message := 'The actuator received a disable request.', level := LogLevel.DEBUG);
			enableRequest := FALSE;
			enable := FALSE;
			timer := disableTime;
			status := ActuatorStatus.DisablePhase;
		ELSIF enabled THEN
			(* End of the enable phase, by feedback or by timeout in no-feedback typology. *)
			enableRequest := FALSE;
			timer := 0;
			status := ActuatorStatus.Enabled;
		END_IF;

	ActuatorStatus.Enabled :
		logger(message := 'Actuator enabled.', level := LogLevel.DEBUG);
		enableRequest := FALSE;

		IF disableRequest THEN
			logger(message := 'The actuator received a disable request.', level := LogLevel.DEBUG);
			enable := FALSE;
			timer := disableTime;
			status := ActuatorStatus.DisablePhase;
		END_IF;

	ActuatorStatus.DisablePhase :
		logger(message := 'Actuator in the disabling phase.', level := LogLevel.DEBUG);

		(* Admissible transition: DisablePhase --> EnablePhase *)
		IF enableRequest THEN
				logger(message := 'The actuator received an enable request.', level := LogLevel.DEBUG);
				disableRequest := FALSE;
				enable := TRUE;
				timer := enableTime;
				status := ActuatorStatus.EnablePhase;
		ELSIF disabled THEN
			(* End of the disable phase, by feedback or by timeout in no-feedback typology. *)
			disableRequest := FALSE;
			timer := 0;
			status := ActuatorStatus.Disabled;
		END_IF;
END_CASE;

(*
 * Diagnostics handler.
 * Generation of diagnosis information and fault signals: Detectable faults in dynamic and static conditions.
 *)
disabledSensorFault := diagnosticsEnable AND (
    (NOT enable AND NOT disabled AND NOT enabled
	OR enable AND disabled AND enabled) AND timeout);
enabledSensorFault := diagnosticsEnable AND (
    (NOT enable AND disabled AND enabled
	OR enable AND NOT disabled AND NOT enabled) AND timeout);
actuatorFault := diagnosticsEnable AND (
    (NOT enable AND NOT disabled AND enabled
	OR enable AND disabled AND NOT enabled) AND timeout);
fault := disabledSensorFault OR enabledSensorFault OR actuatorFault OR externalFault;
(* Log faults *)
IF fault THEN logger(message := 'Fault diagnostics:', level := LogLevel.ERROR); END_IF;
IF disabledSensorFault THEN logger(message := 'Disabled sensor fault.', level := LogLevel.ERROR); END_IF;
IF enabledSensorFault THEN logger(message := 'Enabled sensor fault.', level := LogLevel.ERROR); END_IF;
IF actuatorFault THEN logger(message := 'Actuator fault.', level := LogLevel.ERROR); END_IF;
IF externalFault THEN logger(message := 'External fault (e.g: Motor branch-circuit protection).', level := LogLevel.ERROR); END_IF;

(* Post-elaborations for actuation polymorphism. *)
CASE actuationType OF
	ActuatorActuationType.SingleActuation :
		(* Nothing to do, just use enable *);
	ActuatorActuationType.DoubleActuation :
		disable := NOT enable;
	ActuatorActuationType.DoubleActuationNoRetain :
		enable := enable AND (status = ActuatorStatus.EnablePhase);
		disable := NOT enable AND (status = ActuatorStatus.DisablePhase);
END_CASE;

(* ---- Actuator.st ---- *)
(*
 * Generic binary actuator control system/automata, including mechanisms diagnostics.
 * In nominal conditions, a binary actuator has only two stable equilibrium states: Disabled, Enabled.
 * It also has two unstable transient states: EnablePhase, DisablePhase.
 * The remainder are inadmissible states that must be detected based on timing conditions.
 * Nominal trajectory in the state space, i.e. the evolution of the state in nominal working conditions:
 *     Disabled --> EnablePhase --> Enabled --> DisabledPhase --> back to Disabled
 * Admissible states transitions:
 *     EnablePhase --> DisablePhase, DisablePhase --> EnablePhase
 *
 * Handshake-based actuator control via VAR_IN_OUT.
 * This function block utilizes a Request/Acknowledge (Handshake) mechanism
 * through VAR_IN_OUT variables to manage asynchronous device operations.
 *
 * Usage Logic:
 *  - The caller sets the 'enableRequest' variable to TRUE to initiate the process.
 *  - The FB monitors this variable and attempts to enable the physical device.
 *  - Upon successful activation, the FB internally resets 'enableRequest' to FALSE.
 *
 * Sequencing and diagnostics:
 *  - Sequencing: By monitoring the falling edge of the request variable (Request -> FALSE),
 *    the application logic can deterministically trigger the next step in a sequence
 *    without relying on timers or intermediate state flags.
 *  - Real-Time diagnostics: If the request remains TRUE beyond a defined timeout period,
 *    it indicates a failure in the handshake (e.g., hardware interlock or communication error).
 *    This allows for immediate error detection (machineError) and prevents the
 *    sequence from advancing in an unsafe state.
 *
 * Note:
 * Since the variable is passed by reference (VAR_IN_OUT), both the caller and
 * the FB share the same memory location, ensuring atomic-like synchronization of the command status.
 * This mechanism is used to allow sequencing of the start/stop phases in the presence of a group of devices.
 *
 *)
FUNCTION_BLOCK Actuator
	(* Request/Ack commands *)
	VAR_IN_OUT
	    enableRequest : BOOL;
	    disableRequest : BOOL;
	END_VAR
	VAR_INPUT
		(* Actuator metadata for logging purpose *)
		actuatorId : STRING;
		actuatorName : STRING;
	  	actuationType : ActuatorActuationType;
		feedbackType : ActuatorFeedbackType;
		model : ActuatorModel;
	    operationType : OperatingMode := OperatingMode.Run;
		(* Clock for diagnosis and fault detection under static and dynamic conditions *)
	    clock : BOOL;
		(* Time limit for the enable/disable phase *)
	    enableTime : UINT;
	    disableTime : UINT;
		(* Preset/Reset *)
	    enablePreset : BOOL := FALSE;
	    (* Enable diagnostics *)
	    diagnosticsEnable : BOOL := TRUE;
	END_VAR
	VAR_INPUT
		(* Actuator status sensors *)
	    enabledSensor : BOOL;
	    disabledSensor : BOOL;
		(* External fault signal (e.g. motor branch-circuit protection, thermal relay) *)
		externalFault : BOOL;
		(* Optional parameters  *)
	  	ref : REAL;
	  	feedback : REAL;
	END_VAR
	VAR_OUTPUT
		(* Diagnostics and fault signals *)
	    fault : BOOL;
	    actuatorFault : BOOL;
	    enabledSensorFault : BOOL;
	    disabledSensorFault : BOOL;
	    notInitialized : BOOL;
		(* Logger name for centralized signal management *)
		loggerName : STRING;
	END_VAR
	VAR_OUTPUT
		(* Output signals *)
		enable : BOOL;
	    disable : BOOL;
	END_VAR
	VAR
	    status : ActuatorStatus;
	    timer : UINT;
	    timeout : BOOL;
		(* Internal logical feedback signals (derived from external sensors and/or state + timeout). *)
		enabled : BOOL;
		disabled : BOOL;
		(* Logger facade *)
		logger : LoggerFacade;
	END_VAR

	(* Initialization handler *)
	IF operationType = OperatingMode.Init THEN
		(* Args validation *)
		IF (actuatorId = '' AND actuatorName = '') THEN
			notInitialized := TRUE;
			RETURN;
		END_IF;

		(* Logger facade init *)
		loggerName := concat(concat(concat(actuatorName, '['), actuatorId), ']');
		logger.enable := TRUE; logger.loggerName := loggerName;

		logger(message := 'Actuator initialization.', level := LogLevel.DEBUG);

		(* Pre-elaborations for initialization (polymorphism on feedback typology). *)
		CASE feedbackType OF
			ActuatorFeedbackType.DoubleFeedback :
				enabled := enabledSensor;
				disabled := disabledSensor;

			ActuatorFeedbackType.SingleEnableFeedback :
				enabled := enabledSensor;
				disabled := NOT enabled;

			ActuatorFeedbackType.SingleDisableFeedback :
				disabled := disabledSensor;
				enabled := NOT disabled;

			ActuatorFeedbackType.WithoutFeedback :
				enabled := enablePreset;
				disabled := NOT enabled;
		END_CASE;

		enableRequest := FALSE;
		disableRequest := FALSE;

	    IF enablePreset THEN
			logger(message := 'Actuator preset to enabled status.', level := LogLevel.DEBUG);
			enable := TRUE;
			timer := enableTime;

			IF enabled THEN
				status := ActuatorStatus.Enabled;
				notInitialized := FALSE;
			ELSE
				status := ActuatorStatus.EnablePhase;
	            notInitialized := TRUE;
			END_IF;
	    ELSE
			logger(message := 'Actuator preset to disabled status.', level := LogLevel.DEBUG);
			enable := FALSE;
			timer := disableTime;

			IF disabled THEN
	            status := ActuatorStatus.Disabled;
	            notInitialized := FALSE;
	        ELSE
	            status := ActuatorStatus.DisablePhase;
	            notInitialized := TRUE;
	        END_IF;
		END_IF;
	END_IF;

	IF notInitialized THEN logger(message := 'Actuator not initialized.', level := LogLevel.ERROR); END_IF;

	logger(message := 'Running actuator.', level := LogLevel.DEBUG);

	(* Clock handler for diagnosis oriented timing *)
	IF clock AND (timer > 0) THEN
	    timer := timer - 1;
	END_IF;

	(* Timeout computation *)
	timeout := (timer = 0);

	(* Pre-elaborations for feedback polymorphism. *)
	CASE feedbackType OF
		ActuatorFeedbackType.DoubleFeedback :
			enabled := enabledSensor;
			disabled := disabledSensor;

		ActuatorFeedbackType.SingleDisableFeedback :
			disabled := disabledSensor;
			enabled := (NOT disabled) AND ((status = ActuatorStatus.Enabled)
				OR ((status = ActuatorStatus.EnablePhase) AND timeout));

		ActuatorFeedbackType.SingleEnableFeedback :
			enabled := enabledSensor;
			disabled := (NOT enabled) AND ((status = ActuatorStatus.Disabled)
				OR ((status = ActuatorStatus.DisablePhase) AND timeout));

		ActuatorFeedbackType.WithoutFeedback :
			enabled := (status = ActuatorStatus.Enabled) OR ((status = ActuatorStatus.EnablePhase) AND timeout);
			disabled := (status = ActuatorStatus.Disabled) OR ((status = ActuatorStatus.DisablePhase) AND timeout);
	END_CASE;

	(* Generic actuator FSM implementation. *)
	CASE status OF
		ActuatorStatus.Disabled :
			logger(message := 'Actuator disabled.', level := LogLevel.DEBUG);
			disableRequest := FALSE;

			IF enableRequest THEN
				logger(message := 'The actuator received an enable request.', level := LogLevel.DEBUG);
				enable := TRUE;
				timer := enableTime;
				status := ActuatorStatus.EnablePhase;
			END_IF;

		ActuatorStatus.EnablePhase :
			logger(message := 'Actuator in the enabling phase.', level := LogLevel.DEBUG);

			(* Admissible transition: EnablePhase --> DisablePhase *)
			IF disableRequest THEN
				logger(message := 'The actuator received a disable request.', level := LogLevel.DEBUG);
				enableRequest := FALSE;
				enable := FALSE;
				timer := disableTime;
				status := ActuatorStatus.DisablePhase;
			ELSIF enabled THEN
				(* End of the enable phase, by feedback or by timeout in no-feedback typology. *)
				enableRequest := FALSE;
				timer := 0;
				status := ActuatorStatus.Enabled;
			END_IF;

		ActuatorStatus.Enabled :
			logger(message := 'Actuator enabled.', level := LogLevel.DEBUG);
			enableRequest := FALSE;

			IF disableRequest THEN
				logger(message := 'The actuator received a disable request.', level := LogLevel.DEBUG);
				enable := FALSE;
				timer := disableTime;
				status := ActuatorStatus.DisablePhase;
			END_IF;

		ActuatorStatus.DisablePhase :
			logger(message := 'Actuator in the disabling phase.', level := LogLevel.DEBUG);

			(* Admissible transition: DisablePhase --> EnablePhase *)
			IF enableRequest THEN
					logger(message := 'The actuator received an enable request.', level := LogLevel.DEBUG);
					disableRequest := FALSE;
					enable := TRUE;
					timer := enableTime;
					status := ActuatorStatus.EnablePhase;
			ELSIF disabled THEN
				(* End of the disable phase, by feedback or by timeout in no-feedback typology. *)
				disableRequest := FALSE;
				timer := 0;
				status := ActuatorStatus.Disabled;
			END_IF;
	END_CASE;

	(*
	 * Diagnostics handler.
	 * Generation of diagnosis information and fault signals: Detectable faults in dynamic and static conditions.
	 *)
	disabledSensorFault := diagnosticsEnable AND (
	    (NOT enable AND NOT disabled AND NOT enabled
		OR enable AND disabled AND enabled) AND timeout);
	enabledSensorFault := diagnosticsEnable AND (
	    (NOT enable AND disabled AND enabled
		OR enable AND NOT disabled AND NOT enabled) AND timeout);
	actuatorFault := diagnosticsEnable AND (
	    (NOT enable AND NOT disabled AND enabled
		OR enable AND disabled AND NOT enabled) AND timeout);
	fault := disabledSensorFault OR enabledSensorFault OR actuatorFault OR externalFault;
	(* Log faults *)
	IF fault THEN logger(message := 'Fault diagnostics:', level := LogLevel.ERROR); END_IF;
	IF disabledSensorFault THEN logger(message := 'Disabled sensor fault.', level := LogLevel.ERROR); END_IF;
	IF enabledSensorFault THEN logger(message := 'Enabled sensor fault.', level := LogLevel.ERROR); END_IF;
	IF actuatorFault THEN logger(message := 'Actuator fault.', level := LogLevel.ERROR); END_IF;
	IF externalFault THEN logger(message := 'External fault (e.g: Motor branch-circuit protection).', level := LogLevel.ERROR); END_IF;

	(* Post-elaborations for actuation polymorphism. *)
	CASE actuationType OF
		ActuatorActuationType.SingleActuation :
			(* Nothing to do, just use enable *);
		ActuatorActuationType.DoubleActuation :
			disable := NOT enable;
		ActuatorActuationType.DoubleActuationNoRetain :
			enable := enable AND (status = ActuatorStatus.EnablePhase);
			disable := NOT enable AND (status = ActuatorStatus.DisablePhase);
	END_CASE;
	END_FUNCTION_BLOCK

(* ---- ActuatorGroup.pou ---- *)
(*#-#-#-#-#-#-#-#-#-#---Declaration---#-#-#-#-#-#-#-#-#-#-#-#-#*)

{attribute 'no_assign'}
(*
 * ActuatorGroup - demand-driven staging controller for up to ACTUATOR_GROUP_MAX_SIZE on/off actuators.
 *
 * Inspired by ABB ACH580 PFC (Pump and Fan Control, group 76. See ABB ACH580 drive firmware manual).
 * Progressively starts and stops Actuator FBs to match a varying process demand,
 * with automatic priority rotation (autochange) to balance accumulated run hours.
 *
 * Interface with Actuator FBs
 * The caller declares enableRequests and disableRequests arrays and wires them
 * to the VAR_IN_OUT inputs of each Actuator FB:
 *
 *   pump[i](enableRequest := enReq[i], disableRequest := disReq[i], ...);
 *   grp(enableRequests := enReq, disableRequests := disReq, ...);
 *
 * Both the Actuator and ActuatorGroup share the same array by reference (VAR_IN_OUT).
 * ActuatorGroup writes TRUE to issue a command;
 * the Actuator clears the flag to FALSE as its handshake acknowledgment.
 *
 * IMPORTANT: call each Actuator BEFORE ActuatorGroup in the PLC task so that
 * the actuatorEnabled feedback is current when ActuatorGroup evaluates it.
 *
 * Start / stop staging
 * startPoints[k] (k = 0..actuatorNum-1):
 *   While k actuators are running, if demandSetpoint > startPoints[k] continuously
 *   for startDelay, the next available actuator in the priority order is started (subject to runningNum < maxRunning).
 *   startPoints[0] is the threshold to start the very first actuator (0 → 1).
 *
 * stopPoints[k] (k = 0..actuatorNum-2):
 *   While k+1 actuators are running, if demandSetpoint < stopPoints[k] continuously
 *   for stopDelay, the lowest-priority running actuator is stopped (subject to runningNum > minRunning).
 *   stopPoints[0] is the threshold to stop the last remaining actuator (1 → 0).
 *
 * Demand must hold on one side of the threshold for the full delay before any action is taken.
 * Crossing back resets the timer (anti-cycling hysteresis).
 *
 * Fault / interlock recovery:
 *   Faulted or interlocked actuators are skipped during start selection.
 *   If a running actuator faults and runningNum drops below minRunning, the next
 *   available standby is started immediately (without waiting for startDelay).
 *
 * Autochange:
 * EvenWear: Rotate when the run-hour gap between any two non-faulted
 *           actuators exceeds maxWearImbalance AND demand ≤ autochangeLevel.
 *           The priority array is re-sorted by ascending runHours every cycle;
 *           a physical swap (stop most-used, start least-used) is
 *           triggered only when the imbalance threshold is exceeded.
 * FixedInterval: Rotate every autochangeInterval when demand ≤ autochangeLevel.
 * ExternalTrigger: Rotate on a rising edge of autochangeTrigger when demand ≤ autochangeLevel.
 * AllStopped: Rotate the index array whenever all actuators stop (group
 *             transitions to Disabled). No physical swap is needed because
 *             all are already stopped; the new order takes effect at the next group enable.
 *
 * Rotation sequence (EvenWear / FixedInterval / ExternalTrigger):
 *   1. Stop the selected actuator (disableRequest).
 *   2. Update the priority array (rotate or re-sort).
 *   3. Start the new highest-priority standby actuator (enableRequest).
 *   The group is in the Autochange FSM state for the duration of this sequence.
 *   runningNum briefly drops by 1; set minRunning = 0 if a momentary reduction
 *   is unacceptable and use process-side redundancy instead.
 *)
FUNCTION_BLOCK ActuatorGroup
VAR_EXTERNAL CONSTANT
    (*
	 * Maximum actuators supported. Array bounds in VAR_IN_OUT / VAR_INPUT
     * must match this size exactly in the caller's declaration.
	 *)
    ACTUATOR_GROUP_MAX_SIZE : UINT;
END_VAR
VAR_IN_OUT
    (*
     * Handshake arrays shared with the individual Actuator FBs.
     * ActuatorGroup writes TRUE to command a start or stop.
     * Each Actuator FB clears the flag to FALSE when it accepts the command.
     *)
    enableRequests : ARRAY[1..ACTUATOR_GROUP_MAX_SIZE] OF BOOL;
    disableRequests : ARRAY[1..ACTUATOR_GROUP_MAX_SIZE] OF BOOL;
END_VAR
VAR_INPUT
	(* Actuator group metadata for logging purpose *)
	actuatorGroupId : STRING;
	actuatorGroupName : STRING;

    (* Topology *)
    (* Total actuators declared in the group. Must be 1..ACTUATOR_GROUP_MAX_SIZE. *)
    actuatorNum : UINT := 1;
    (* Minimum actuators to keep running simultaneously (0 = allow full stop). *)
    minRunning : UINT := 1;
    (* Maximum actuators allowed running simultaneously. *)
    maxRunning : UINT := 1;

    (* Process demand *)
    (* Demand setpoint in percent (0.0 ... 100.0). Drives all start/stop decisions. *)
    demandSetpoint : REAL;

    (*
     * Start / stop thresholds.
     * startPoints[k]: demand level that triggers starting the (k+1)-th
     * actuator while exactly k are currently running (k = 0..actuatorNum-1).
     * startPoints[0] = threshold to start the first actuator (0 → 1).
	 *)
    startPoints : ARRAY[0..7] OF REAL;
    (*
     * stopPoints[k]: demand level below which the (k+1)-th running actuator is stopped (k = 0..actuatorNum-2).
     * stopPoints[0] = threshold to stop the last actuator (1 → 0).
     *)
    stopPoints : ARRAY[0..7] OF REAL;
    (* Demand must stay above startPoints[k] for this long before a start. *)
    startDelay : TIME := T#10s;
    (* Demand must stay below stopPoints[k] for this long before a stop. *)
    stopDelay : TIME := T#10s;

    (* Autochange *)
    autochange : ActuatorGroupAutochange := ActuatorGroupAutochange.None;
    (* Period for FixedInterval rotation. *)
    autochangeInterval : TIME := T#1h;
    (*
     * Max allowed run-hour gap between most-used and least-used actuator
     * before EvenWear triggers a swap (hours, e.g. 72.0 for 3 days).
     *)
    maxWearImbalance : REAL := 72.0;
    (* Autochange is only triggered when demandSignal ≤ autochangeLevel. *)
    autochangeLevel : REAL := 100.0;
    (* Rising edge triggers an immediate autochange (ExternalTrigger mode). *)
    autochangeTrigger : BOOL;

    (* Per-actuator feedback *)
    (*
     * Map actuatorEnabled[i] from Actuator[i].enable (TRUE in EnablePhase
     * AND Enabled states - i.e., the actuator is active or starting up).
     *)
    actuatorEnabled : ARRAY[1..ACTUATOR_GROUP_MAX_SIZE] OF BOOL;
    (* Map actuatorFault[i] from Actuator[i].fault. *)
    actuatorFault : ARRAY[1..ACTUATOR_GROUP_MAX_SIZE] OF BOOL;
    (* External maintenance / hardware interlock flag per actuator. *)
    actuatorInterlocked : ARRAY[1..ACTUATOR_GROUP_MAX_SIZE] OF BOOL;
    (* Cumulative run time in hours, maintained by the caller (e.g., a REAL counter incremented by 1/3600 each second). *)
    runHours : ARRAY[1..ACTUATOR_GROUP_MAX_SIZE] OF REAL;

    (* Group commands *)
    (*
      * Rising edge (FALSE→TRUE) starts the group (Disabled → Running).
      * Cleared by the FB when the transition is accepted.
     *)
    groupEnable : BOOL;
    (*
     * Rising edge (FALSE→TRUE) stops the group (Running → Stopping → Disabled).
     * Cleared by the FB when the transition is accepted.
     *)
    groupDisable : BOOL;
END_VAR
VAR_OUTPUT
    (* Current group FSM state. *)
    status : ActuatorGroupStatus := ActuatorGroupStatus.Disabled;
    (* Actuators neither faulted nor interlocked (available for use). *)
    availableNum : UINT;
    (* Actuators currently active (Enabled or EnablePhase). *)
    runningNum : UINT;
    (* TRUE when nAvailable < actuatorNum (one or more offline/faulted). *)
    degraded : BOOL;
    (* TRUE when a fault has left runningNum below minRunning. *)
    underMinimum : BOOL;
    (* TRUE when configuration inputs are invalid. *)
    invalidConfig : BOOL;
    (* TRUE while an autochange rotation is in progress. *)
    autochangeActive : BOOL;
	(* Logger name for centralized signal management *)
	loggerName : STRING;
END_VAR
VAR
    (* Internal FSM state *)
    internalStatus : ActuatorGroupStatus := ActuatorGroupStatus.Disabled;

    (* Priority order *)
    (*
	 * sortedIdx[1] = first to start / last to stop.
     * sortedIdx[actuatorNum] = last to start / first to stop.
     * Initialised to [1, 2, … actuatorNum] on the first call.
     *)
    sortedIdx : ARRAY[1..ACTUATOR_GROUP_MAX_SIZE] OF UINT;

    (* Autochange bookkeeping *)
    autochangeStep : UINT; (* 0 = idle, 1 = stopping old, 2 = starting new *)
    autochangeStopIdx : UINT; (* physical actuator slot being stopped *)
    autochangeStartIdx : UINT; (* physical actuator slot being started *)
    autochangeTrigOld : BOOL; (* previous cycle value for edge detection *)

    (* Timer signals *)
    (* Computed each cycle in the FSM; passed to TON FBs at the bottom. *)
    startTimerTrig : BOOL;
    stopTimerTrig : BOOL;
    autochangeTimerTrig : BOOL;
    startTimer : TON;
    stopTimer : TON;
    autochangeTimer : TON;

    (* Loop temporaries *)
    i, j, tempIdx : UINT;
    swapped : BOOL;
    minHoursIdx : UINT;
    maxHoursIdx : UINT;
	(* Logger facade *)
	logger : LoggerFacade;
	init : BOOL;
END_VAR

(*#-#-#-#-#-#-#-#-#-#---Implementation---#-#-#-#-#-#-#-#-#-#-#-#-#*)

(* Init *)
IF NOT init THEN
	IF (actuatorGroupId = '' AND actuatorGroupName = '') THEN
		invalidConfig := TRUE;
		RETURN;
	END_IF;

	(* Logger facade init *)
	loggerName := concat(concat(concat(actuatorGroupName, '['), actuatorGroupId), ']');
	logger.enable := TRUE; logger.loggerName := loggerName;
	init := TRUE;
END_IF;

logger(message := 'Running actuator group.', level := LogLevel.DEBUG);

(* Args validation *)
invalidConfig := (actuatorNum < 1) OR (actuatorNum > ACTUATOR_GROUP_MAX_SIZE)
	OR (minRunning < 0) OR (maxRunning < 1)
    OR (minRunning > maxRunning)
    OR (maxRunning > actuatorNum);
IF invalidConfig THEN
    status := ActuatorGroupStatus.Disabled;
    RETURN;
END_IF;

(* Init priority index on first call or when actuatorNum grows.
 * Valid slot indices are 1..actuatorNum; 0 is the zero-initialised
 * default and is never a valid value, so a zero entry always means the slot
 * has not been assigned yet. This allows the group to be reconfigured at
 * run-time with a larger actuatorNum without re-setting existing order. *)
FOR i := 1 TO actuatorNum DO
    IF sortedIdx[i] = 0 THEN
        sortedIdx[i] := i;
    END_IF;
END_FOR;

(* Count available and active actuators (every cycle) *)
availableNum := 0;
runningNum   := 0;
FOR i := 1 TO actuatorNum DO
    IF NOT actuatorFault[i] AND NOT actuatorInterlocked[i] THEN
        availableNum := availableNum + 1;
    END_IF;
    IF actuatorEnabled[i] THEN
        runningNum := runningNum + 1;
    END_IF;
END_FOR;
degraded := (availableNum < actuatorNum);
underMinimum := (internalStatus = ActuatorGroupStatus.Running) AND (runningNum < minRunning);

(* EvenWear priority re-sort (runs every cycle when EvenWear is active) *)
(*
 * Sort sortedIdx[1..actuatorNum] by ascending runHours so that the actuator
 * with the fewest cumulative hours is always started first.
 * Faulted / interlocked actuators are bubbled to the end of the array so they
 * are naturally skipped when the start/stop logic scans the priority order.
 *
 * The sort runs every cycle in Running and Autochange states.  For other
 * autochange modes the order is updated only by explicit rotation steps.
 *)
IF autochange = ActuatorGroupAutochange.EvenWear
        AND (internalStatus = ActuatorGroupStatus.Running
		OR internalStatus = ActuatorGroupStatus.Autochange) THEN
    FOR i := 1 TO actuatorNum - 1 DO
        swapped := FALSE;
        FOR j := 1 TO actuatorNum - i DO
            (* Push faulted / interlocked slots to the end *)
            IF (actuatorFault[sortedIdx[j]] OR actuatorInterlocked[sortedIdx[j]])
                    AND NOT (actuatorFault[sortedIdx[j + 1]] OR actuatorInterlocked[sortedIdx[j + 1]])
               (* Among healthy slots: sort by ascending run hours *)
               OR (NOT (actuatorFault[sortedIdx[j]] OR actuatorInterlocked[sortedIdx[j]])
                   AND NOT (actuatorFault[sortedIdx[j + 1]] OR actuatorInterlocked[sortedIdx[j + 1]])
                   AND runHours[sortedIdx[j]] > runHours[sortedIdx[j + 1]]) THEN
                tempIdx := sortedIdx[j];
                sortedIdx[j] := sortedIdx[j + 1];
                sortedIdx[j + 1] := tempIdx;
                swapped := TRUE;
            END_IF;
        END_FOR;

        IF NOT swapped THEN EXIT; END_IF;
    END_FOR;
END_IF;

(* Timer signal defaults (overridden by the Running state block) *)
startTimerTrig := FALSE;
stopTimerTrig := FALSE;
(*
 * AutochangeTimer only accumulates while Running - interval is operating time, not wall time.
 * The Running state sets this FALSE for one cycle after .Q fires to reset the period.
 *)
autochangeTimerTrig := (autochange = ActuatorGroupAutochange.FixedInterval)
	AND (internalStatus = ActuatorGroupStatus.Running);

(* Main FSM *)
CASE internalStatus OF
    (* Disabled: no actuators running. Wait for groupEnable. *)
    ActuatorGroupStatus.Disabled :
        groupDisable := FALSE;
        autochangeActive := FALSE;
        autochangeStep := 0;

        IF groupEnable AND availableNum >= minRunning THEN
			logger(message := 'Actuator group running.', level := LogLevel.DEBUG);
            groupEnable := FALSE;
            internalStatus := ActuatorGroupStatus.Running;
        ELSIF groupEnable AND availableNum < minRunning THEN
            (* Not enough actuators available - refuse enable *)
            groupEnable := FALSE;
        END_IF;

    (* Running: demand-driven start / stop of individual actuators. *)
    ActuatorGroupStatus.Running :
        groupEnable := FALSE;
        autochangeActive := FALSE;

        (* Disable command: transition to Stopping *)
        IF groupDisable THEN
            groupDisable := FALSE;
            FOR i := 1 TO actuatorNum DO
                IF actuatorEnabled[i] THEN
                    disableRequests[i] := TRUE;
                END_IF;
                enableRequests[i] := FALSE; (* Cancel pending starts *)
            END_FOR;

			internalStatus := ActuatorGroupStatus.Stopping;
			logger(message := 'Actuator group stopping.', level := LogLevel.DEBUG);
        ELSE
            (* Fault recovery: restore minRunning immediately (no delay). *)
            (*
             * If a running actuator has faulted and runningNum < minRunning,
             * start the next available standby without waiting for startDelay.
             * Only one start per cycle to avoid over-driving the process.
             *)
            IF runningNum < minRunning THEN
                FOR i := 1 TO actuatorNum DO
                    IF NOT actuatorEnabled[sortedIdx[i]]
							AND NOT actuatorFault[sortedIdx[i]]
                            AND NOT actuatorInterlocked[sortedIdx[i]]
                            AND NOT enableRequests[sortedIdx[i]] THEN
                        enableRequests[sortedIdx[i]] := TRUE;
                        EXIT;
                    END_IF;
                END_FOR;
            END_IF;

            (* Normal start: add the next unit when demand is high. *)
            (*
             * Check startPoints[runningNum]: the threshold to go from runningNum to runningNum+1 active actuators.
			 * Array index matches the current running count (ABB 76.30: "velocity to start auxiliary k").
             * The timer runs as long as the condition holds; it resets
             * automatically if demand drops back below the threshold.
             *)
            IF runningNum >= minRunning AND runningNum < maxRunning
                    AND runningNum <= actuatorNum - 1 THEN
                startTimerTrig := (demandSetpoint > startPoints[runningNum]);
                IF startTimer.Q THEN
                    FOR i := 1 TO actuatorNum DO
                        IF NOT actuatorEnabled[sortedIdx[i]]
                                AND NOT actuatorFault[sortedIdx[i]]
                                AND NOT actuatorInterlocked[sortedIdx[i]]
                                AND NOT enableRequests[sortedIdx[i]] THEN
                            enableRequests[sortedIdx[i]] := TRUE;
                            EXIT;
                        END_IF;
                    END_FOR;

                    startTimerTrig := FALSE; (* Reset timer after issuing start *)
                END_IF;
            END_IF;

            (* Normal stop: remove the last unit when demand is low. *)
            (*
             * Check stopPoints[runningNum - 1]: the threshold to go from runningNum
             * to runningNum-1 active actuators. Index runningNum-1 is always >= 0
             * because runningNum > minRunning >= 0. The last actuator in the
             * sorted order (highest index) is stopped first (LIFO principle).
             *)
            IF runningNum > minRunning
                    AND runningNum - 1 <= actuatorNum - 1 THEN
                stopTimerTrig := (demandSetpoint < stopPoints[runningNum - 1]);
                IF stopTimer.Q THEN
                    FOR i := actuatorNum TO 1 BY -1 DO
                        IF actuatorEnabled[sortedIdx[i]]
                                AND NOT disableRequests[sortedIdx[i]] THEN
                            disableRequests[sortedIdx[i]] := TRUE;
                            EXIT;
                        END_IF;
                    END_FOR;

                    stopTimerTrig := FALSE; (* Reset timer after issuing stop *)
                END_IF;
            END_IF;

            (* Autochange trigger evaluation *)
            IF autochange <> ActuatorGroupAutochange.None
                    AND autochange <> ActuatorGroupAutochange.AllStopped
                    AND runningNum > 0
                    AND demandSetpoint <= autochangeLevel THEN

                CASE autochange OF
                    (* EvenWear *)
                    ActuatorGroupAutochange.EvenWear :
                        (*
                         * Find the running actuator with the most hours and the
                         * standby actuator with the fewest hours.
						 * Trigger a swap when the imbalance exceeds maxWearImbalance (hours).
                         *)
                        minHoursIdx := 0; maxHoursIdx := 0;
                        FOR i := 1 TO actuatorNum DO
                            IF NOT actuatorFault[i] AND NOT actuatorInterlocked[i] THEN
                                IF minHoursIdx = 0 THEN
                                    minHoursIdx := i;
                                ELSIF runHours[i] < runHours[minHoursIdx] THEN
                                    minHoursIdx := i;
                                END_IF;
                                IF maxHoursIdx = 0 THEN
                                    maxHoursIdx := i;
                                ELSIF runHours[i] > runHours[maxHoursIdx] THEN
                                    maxHoursIdx := i;
                                END_IF;
                            END_IF;
                        END_FOR;

                        IF minHoursIdx > 0 AND maxHoursIdx > 0
                                AND minHoursIdx <> maxHoursIdx
                                AND (runHours[maxHoursIdx] - runHours[minHoursIdx]) > maxWearImbalance
                                AND actuatorEnabled[maxHoursIdx]
                                AND NOT actuatorEnabled[minHoursIdx]
                                AND NOT actuatorFault[minHoursIdx]
                                AND NOT actuatorInterlocked[minHoursIdx] THEN
                            autochangeStopIdx := maxHoursIdx;
                            autochangeStartIdx := 0; (* Resolved in Autochange step 1 *)
                            autochangeStep := 1;
                            disableRequests[autochangeStopIdx] := TRUE;
                            internalStatus := ActuatorGroupStatus.Autochange;
                        END_IF;

                    (* FixedInterval *)
                    ActuatorGroupAutochange.FixedInterval :
                        IF autochangeTimer.Q THEN
                            (* Select the lowest-priority running actuator to stop *)
                            autochangeStopIdx := 0;
                            FOR i := actuatorNum TO 1 BY -1 DO
                                IF actuatorEnabled[sortedIdx[i]] THEN
                                    autochangeStopIdx := sortedIdx[i];
                                    EXIT;
                                END_IF;
                            END_FOR;

                            IF autochangeStopIdx > 0 THEN
                                autochangeStep := 1;
                                disableRequests[autochangeStopIdx] := TRUE;
                                internalStatus := ActuatorGroupStatus.Autochange;
                            END_IF;

                            (* Reset the interval timer regardless of whether we swapped *)
                            autochangeTimerTrig := FALSE;
                        END_IF;

                    (* ExternalTrigger *)
                    ActuatorGroupAutochange.ExternalTrigger :
                        IF autochangeTrigger AND NOT autochangeTrigOld THEN
                            autochangeStopIdx := 0;

                            FOR i := actuatorNum TO 1 BY -1 DO
                                IF actuatorEnabled[sortedIdx[i]] THEN
                                    autochangeStopIdx := sortedIdx[i];
                                    EXIT;
                                END_IF;
                            END_FOR;

                            IF autochangeStopIdx > 0 THEN
                                autochangeStep := 1;
                                disableRequests[autochangeStopIdx] := TRUE;
                                internalStatus := ActuatorGroupStatus.Autochange;
                            END_IF;
                        END_IF;
                END_CASE;
            END_IF;
        END_IF; (* groupDisable / else *)

    (* Stopping: wait for all actuators to reach disabled state. *)
    ActuatorGroupStatus.Stopping :
        IF runningNum = 0 THEN
            (*
             * AllStopped autochange: rotate the priority order now that all
             * actuators are off.  The new order takes effect at the next
             * groupEnable.  No physical swap is needed (all already stopped).
             *)
            IF autochange = ActuatorGroupAutochange.AllStopped THEN
                tempIdx := sortedIdx[1];
                FOR i := 1 TO actuatorNum - 1 DO
                    sortedIdx[i] := sortedIdx[i + 1];
                END_FOR;
                sortedIdx[actuatorNum] := tempIdx;
            END_IF;

            internalStatus := ActuatorGroupStatus.Disabled;
        END_IF;

    (*
     * Autochange: sequential stop / rotate / start.
     *
     * Step 1 - wait for the old actuator to stop.
     * Step 2 - start the new highest-priority standby.
     *)
    ActuatorGroupStatus.Autochange :
		logger(message := 'Actuator group autochange.', level := LogLevel.DEBUG);
        autochangeActive := TRUE;
        groupEnable := FALSE;

        (* Disable command during autochange: abort and go to Stopping *)
        IF groupDisable THEN
            groupDisable := FALSE;

            FOR i := 1 TO actuatorNum DO
                IF actuatorEnabled[i] THEN disableRequests[i] := TRUE; END_IF;
                enableRequests[i] := FALSE;
            END_FOR;

            internalStatus := ActuatorGroupStatus.Stopping;
        ELSE
            CASE autochangeStep OF
                1 : (* Waiting for the old actuator to finish stopping *)
                    IF NOT actuatorEnabled[autochangeStopIdx] THEN
                        (*
                         * Old actuator is now off.  Update the priority order:
                         * - FixedInterval / ExternalTrigger: rotate the stopped
                         *   actuator from its current position to the end of the
                         *   array so it is the last to be started next time.
                         * - EvenWear: the continuous sort (above) already
                         *   maintains the correct order; no manual rotation needed.
                         *)
                        IF autochange = ActuatorGroupAutochange.FixedInterval
                                OR autochange = ActuatorGroupAutochange.ExternalTrigger THEN
                            FOR i := 1 TO actuatorNum DO
                                IF sortedIdx[i] = autochangeStopIdx THEN
                                    FOR j := i TO actuatorNum - 1 DO
                                        sortedIdx[j] := sortedIdx[j + 1];
                                    END_FOR;
                                    sortedIdx[actuatorNum] := autochangeStopIdx;
                                    EXIT;
                                END_IF;
                            END_FOR;
                        END_IF;

                        (* Find the highest-priority standby to start *)
                        autochangeStartIdx := 0;
                        FOR i := 1 TO actuatorNum DO
                            IF NOT actuatorEnabled[sortedIdx[i]]
                                    AND NOT actuatorFault[sortedIdx[i]]
                                    AND NOT actuatorInterlocked[sortedIdx[i]] THEN
                                autochangeStartIdx := sortedIdx[i];
                                EXIT;
                            END_IF;
                        END_FOR;

                        IF autochangeStartIdx > 0 THEN
                            enableRequests[autochangeStartIdx] := TRUE;
                            autochangeStep := 2;
                        ELSE
                            (* No standby available; return without starting a replacement *)
                            autochangeStep := 0;
                            internalStatus := ActuatorGroupStatus.Running;
                        END_IF;
                    END_IF;

                2 : (* Waiting for the new actuator to reach enabled state *)
                    IF actuatorEnabled[autochangeStartIdx] THEN
                        autochangeStep := 0;
                        internalStatus := ActuatorGroupStatus.Running;
                    END_IF;
            END_CASE;
        END_IF;
END_CASE; (* internalStatus *)

(* Unconditional timer calls (once per cycle, after FSM) *)
(*
 * startTimer / stopTimer: anti-cycling guards for demand-driven start/stop.
 *   IN is driven by the Running state logic above.
 *   IN goes FALSE automatically when:
 *     - demand reverses (anti-cycling, timer resets before Q fires), or
 *     - the FSM exits Running state (timer.IN defaults to FALSE above), or
 *     - a start/stop action is taken (timer.IN forced FALSE in the action).
 *
 * autochangeTimer: fixed-interval rotation period. Runs whenever
 *   autochange = FixedInterval, regardless of FSM state.  The timer is
 *   reset by setting autochangeTimer_IN := FALSE for one cycle (done in
 *   the Running state when the timer fires).
 *)
startTimer(IN := startTimerTrig, PT := startDelay);
stopTimer(IN := stopTimerTrig, PT := stopDelay);
autochangeTimer(IN := autochangeTimerTrig, PT := autochangeInterval);

(* Rising-edge latch - update after all logic that reads it *)
autochangeTrigOld := autochangeTrigger;

(* Status output *)
status := internalStatus;
